TYPE "PLCtoMES_ProcessData"
VERSION : 0.1
   STRUCT
      SubResult : Byte;
      SubUSL : Real;
      SubResultValue : Real;
      SubLSL : Real;
   END_STRUCT;

END_TYPE

